Staubli VAL3: power.pgx

public program power(bool bState (dimensions=1), bool& bFlag[] (dimensions=1))
begin
  switch bState
    case false
      disablePower()
      bFlag=true
    break
    case true
      enablePower()
      if (watch(isPowered(),3)==false)
        bFlag=false
      else
        bFlag=true
      endIf
    break
  endSwitch
end
